// TIA Portal V20 export
// export: Created 2026-04-11T06:02:29.948118Z, ExportSetting WithDefaults, DisplayName Totally Integrated Automation Portal, DisplayVersion V20, DisplayName TIA Portal Openness, DisplayVersion V20, DisplayName TIA Portal Version Control Interface, DisplayVersion V20, DisplayName STEP 7 Professional, DisplayVersion V20, DisplayName STEP 7 Safety, DisplayVersion V20, DisplayName WinCC Basic/Comfort/Advanced, DisplayVersion V20, DisplayName WinCC Unified, DisplayVersion V20
TYPE "udtError_AnalogInput"
// stored: IsFailsafeCompliant false
   STRUCT
      LowLowAlarm { ExternalWritable := 'False'} : Bool;   // Value below low low set point
      HighHighAlarm { ExternalWritable := 'False'} : Bool;   // Value above high high set point
      Invalid { ExternalWritable := 'False'} : Bool;   // Invalid input valid
   END_STRUCT;
END_TYPE
